RoboDK station: Drawing with a robot.rdk

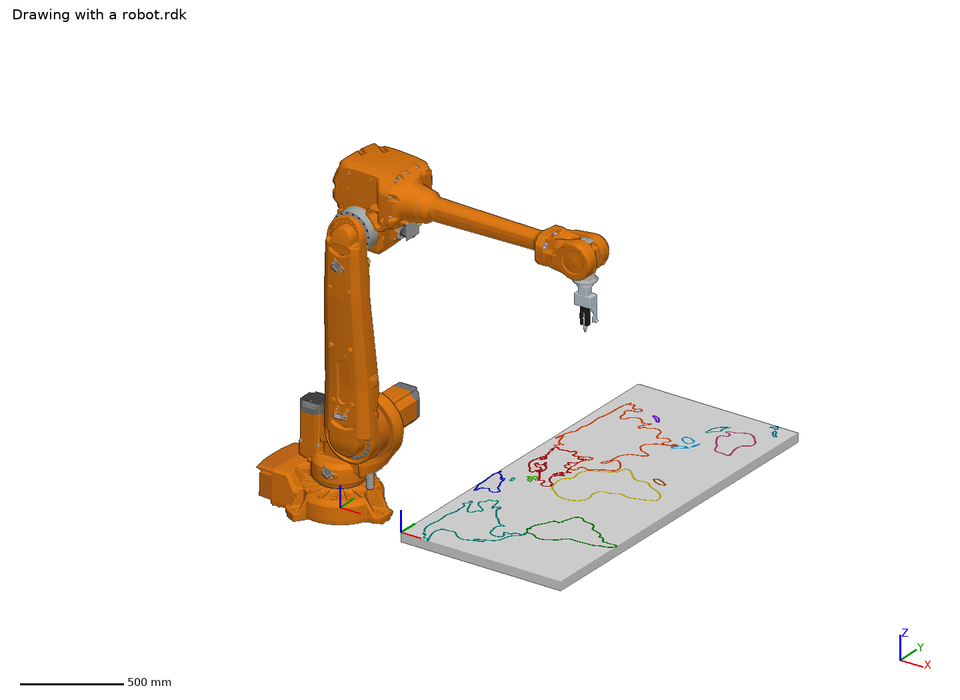
[picture v0: the station drawn from its stored meshes, robots at their saved joint values, targets as dots, program paths as lines]
Station Example 3 - Drawing with a robot. Poses are relative to the parent item; angles as X-Y-Z fixed-axis rotations.
  - Python program Robot paint (listed below)
  - frame ABB IRB 4600-20/2.50 Base at (0, 0, 0) mm
    - robot ABB IRB 4600-20/2.50: 6 axes, payload 20 kg, reach 2500 mm, repeatability 0.05 mm, weight 412 kg
        modified DH rows (alpha deg, a mm, theta deg, d mm): 0, 0, 0, 495; -90, 175, -90, 0; 0, 1095, 0, 0; -90, 175, 0, 1270; 90, 0, 0, 0; -90, 0, 180, 135
        joint limits [-180, -90, -180, -400, -120, -400] to [180, 150, 75, 400, 120, 400]; home [0, 0, 0, 0, 90, 0]; saved at [0, 0, 0, 0, 90, 0]
      - tool Tool, TCP at (0, 0, 283) mm, size 100 x 89.2 x 281.5 mm
    - object pixel at (0, 0, 0) mm, size 10 x 10 x 1 mm
    - frame Frame draw at (1016.5, -940.57, 525.71) mm
      - object Blackboard 250mm at (0, 0, 0) mm, size 250 x 250 x 50 mm
      - object Board & image at (0, 0, 0) mm, size 955.9 x 2016.4 x 51 mm

--- Python program Robot paint ---
from robolink import *    # API to communicate with RoboDK
from robodk import *      # robodk robotics toolbox

import sys
import os
import re

PIXELS_AS_OBJECTS = False    # Set to True to generate PDF or HTML simulations that include the drawn path
TCP_KEEP_TANGENCY = False    # Set to True to keep the tangency along the path
SIZE_BOARD = [1000, 2000]     # Size of the image. The image will be scaled keeping its aspect ratio
MM_X_PIXEL = 10             # in mm. The path will be cut depending on the pixel size. If this value is changed it is recommended to scale the pixel object
IMAGE_FILE = 'World map.svg'             # Path of the SVG image, it can be relative to the current RDK station

#--------------------------------------------------------------------------------
# function definitions:

def point2D_2_pose(point, tangent):
    """Converts a 2D point to a 3D pose in the XY plane including rotation being tangent to the path"""
    return transl(point.x, point.y, 0)*rotz(tangent.angle())

def svg_draw_quick(svg_img, board, pix_ref):
    """Quickly shows the image result without checking the robot movements."""
    RDK.Render(False)
    count = 0
    for path in svg_img:
        count = count + 1
        # use the pixel reference to set the path color, set pixel width and copy as a reference
        pix_ref.Recolor(path.fill_color)
        if PIXELS_AS_OBJECTS:
            pix_ref.Copy()
        np = path.nPoints()
        print('drawing path %i/%i' % (count, len(svg_img)))
        for i in range(np):
            p_i = path.getPoint(i)
            v_i = path.getVector(i)

            # Reorient the pixel object along the path
            pt_pose = point2D_2_pose(p_i, v_i)

            # add the pixel geometry to the drawing board object, at the calculated pixel pose
            if PIXELS_AS_OBJECTS:
                board.Paste().setPose(pt_pose)
            else:
                board.AddGeometry(pix_ref, pt_pose)

    RDK.Render(True)

def svg_draw_robot(svg_img, board, pix_ref, item_frame, item_tool, robot):
    """Draws the image with the robot. It is slower that svg_draw_quick but it makes sure that the image can be drawn with the robot."""

    APPROACH = 100  # approach distance in MM for each path
    home_joints = robot.JointsHome().tolist() #[0,0,0,0,90,0] # home joints, in deg
    if abs(home_joints[4]) < 5:
        home_joints[4] = 90.0

    robot.setPoseFrame(item_frame)
    robot.setPoseTool(item_tool)
    robot.MoveJ(home_joints)

    # get the target orientation depending on the tool orientation at home position
    orient_frame2tool = invH(item_frame.Pose())*robot.SolveFK(home_joints)*item_tool.Pose()
    orient_frame2tool[0:3,3] = Mat([0,0,0])
    # alternative: orient_frame2tool = roty(pi)

    for path in svg_img:
        # use the pixel reference to set the path color, set pixel width and copy as a reference
        print('Drawing %s, RGB color = [%.3f,%.3f,%.3f]'%(path.idname, path.fill_color[0], path.fill_color[1], path.fill_color[2]))
        pix_ref.Recolor(path.fill_color)
        if PIXELS_AS_OBJECTS:
            pix_ref.Copy()
        np = path.nPoints()

        # robot movement: approach to the first target
        p_0 = path.getPoint(0)
        target0 = transl(p_0.x, p_0.y, 0)*orient_frame2tool
        target0_app = target0*transl(0,0,-APPROACH)
        robot.MoveL(target0_app)

        #if TCP_KEEP_TANGENCY:
        #    joints_now = robot.Joints().tolist()
        #    joints_now[5] = -180
        #    robot.MoveJ(joints_now)
        RDK.RunMessage('Drawing %s' % path.idname);
        RDK.RunProgram('SetColorRGB(%.3f,%.3f,%.3f)' % (path.fill_color[0], path.fill_color[1], path.fill_color[2]))
        for i in range(np):
            p_i = path.getPoint(i)
            v_i = path.getVector(i)

            pt_pose = point2D_2_pose(p_i, v_i)

            if TCP_KEEP_TANGENCY:
                #moving the tool along the path (axis 6 may reach its limits)
                target = pt_pose*orient_frame2tool
            else:
                #keep the tool orientation constant
                target = transl(p_i.x, p_i.y, 0)*orient_frame2tool

            # Move the robot to the next target
            robot.MoveL(target)

            # create a new pixel object with the calculated pixel pose
            if PIXELS_AS_OBJECTS:
                board.Paste().setPose(pt_pose)
            else:
                board.AddGeometry(pix_ref, pt_pose)

        target_app = target*transl(0,0,-APPROACH)
        robot.MoveL(target_app)

    robot.MoveL(home_joints)

#--------------------------------------------------------------------------------
# Program start
RDK = Robolink()

# locate and import the svgpy module
# Old versions of RoboDK required adding required paths to the process path
# New versions of RoboDK automatically add the current folder to the path (after 4.2.2)
path_stationfile = RDK.getParam('PATH_OPENSTATION')
#sys.path.append(os.path.abspath(path_stationfile)) # temporary add path to import station modules
#print(os.getcwd())
#print(os.environ['PYTHONPATH'].split(os.pathsep))
#print(os.environ['PATH'].split(os.pathsep))


from svgpy.svg import *

# select the file to draw
svgfile = IMAGE_FILE
if len(svgfile) == 0:
    svgfile = getOpenFile()
elif not FileExists(svgfile):
    svgfile = path_stationfile + '/' + svgfile

#svgfile = path_stationfile + '/World map.svg'
#svgfile = path_stationfile + '/RoboDK text.svg'

# import the SVG file
svgdata = svg_load(svgfile)

IMAGE_SIZE = Point(SIZE_BOARD[0],SIZE_BOARD[1])   # size of the image in MM
svgdata.calc_polygon_fit(IMAGE_SIZE, MM_X_PIXEL)
size_img = svgdata.size_poly()  # returns the size of the current polygon

# get the robot, frame and tool objects
robot = RDK.ItemUserPick('', ITEM_TYPE_ROBOT)
framedraw = RDK.Item('Frame draw')
tooldraw = RDK.Item('Tool')

# get the pixel reference to draw
pixel_ref = RDK.Item('pixel')

# delete previous image if any
image = RDK.Item('Board & image')
if image.Valid() and image.Type() == ITEM_TYPE_OBJECT: image.Delete()

# make a drawing board base on the object reference "Blackboard 250mm"
board_1m = RDK.Item('Blackboard 250mm')
board_1m.Copy()
board_draw = framedraw.Paste()
board_draw.setVisible(True, False)
board_draw.setName('Board & image')
board_draw.Scale([size_img.x/250, size_img.y/250, 1]) # adjust the board size to the image size (scale)

pixel_ref.Copy()

# quickly show the final result without checking the robot movements:
#svg_draw_quick(svgdata, board_draw, pixel_ref)

# draw the image with the robot:
svg_draw_robot(svgdata, board_draw, pixel_ref, framedraw, tooldraw, robot)
